TYPE Tank_Io_In :
STRUCT
	bEnable			: BOOL;
	fLevel			: REAL;
END_STRUCT
END_TYPE

(* stored: Version 1.1.0.1
   DUT Tank_Io_In: Id {b91ccb76-0f8a-4c0c-9443-4a956ae894a9} *)
